PROGRAM MAIN
VAR
END_VAR

//IO.bOutput := HMI.bContactor;
HMI.iTemperatureDisplayValue := IO.iInput/10;
//Temperature Control state
IF HMI.bTemperatureControlSwitch = 1 THEN
	HMI.sTemperatureControlState := 'AUTO';
END_IF
IF HMI.bTemperatureControlSwitch = 0 THEN
	HMI.sTemperatureControlState := 'MAN';
END_IF

END_PROGRAM

(* stored: Version 1.1.0.1, ProductVersion 3.1.4024.9
   POU MAIN: Id {dec5b1ca-8e16-4f49-8efb-57a750654862}, SpecialFunc None *)
